// TIA Portal V17 export
// export: Created 2022-07-20T06:59:52.0228189Z, ExportSetting WithDefaults, DisplayName Totally Integrated Automation Portal, DisplayVersion V17, DisplayName TIA Portal Openness, DisplayVersion V17, DisplayName TIA Portal Version Control Interface, DisplayVersion V17, DisplayName SINAMICS Startdrive Advanced, DisplayVersion V17, DisplayName SINAMICS Startdrive G130, G150, S120, S150, SINAMICS MV, S210, DisplayVersion V17, DisplayName SINAMICS Startdrive G110M, G120, G120C, G120D, G120P, G115D, DisplayVersion V17, DisplayName STEP 7 Professional, DisplayVersion V17, DisplayName STEP 7 Safety, DisplayVersion V17, DisplayName WinCC Advanced, DisplayVersion V17
FUNCTION_BLOCK "FB10400_APCMotor"   // FB10400, LAD
{ S7_Optimized_Access := 'TRUE' }
VERSION : 0.1
// stored: AutoNumber false, IsIECCheckEnabled false, IsRetainMemResEnabled false, MemoryReserve 100, SetENOAutomatically false, UDAEnableTagReadback false
   VAR_INPUT
      ToAxis : TO_PositioningAxis;
      HomingSensor : Bool;
      RequestDirectHoming : Bool;
      RequestSensorHoming : Bool;
      RequestTorqueHoming : Bool;
      RequestGoToAbsolutePosition_1 : Bool;
      RequestGoToAbsolutePosition_2 : Bool;
      RequestGoToAbsolutePosition_3 : Bool;
      RequestGoToAbsolutePosition_4 : Bool;
      RequestGoToAbsolutePosition_5 : Bool;
      RequestGoToAbsolutePosition_6 : Bool;
      RequestGoToAbsolutePosition_7 : Bool;
      RequestGoToAbsolutePosition_8 : Bool;
      RequestGoToAbsolutePosition_9 : Bool;
      RequestGoToAbsolutePosition_10 : Bool;
      RequestGoToRelativePosition : Bool;
      RequestJogForward : Bool;
      RequestJogBackward : Bool;
      RequestStop : Bool;
      RequestFastStop : Bool;
      RequestAcknowledge : Bool;
      AbsolutePosition_1 : LReal;
      AbsolutePosition_2 : LReal;
      AbsolutePosition_3 : LReal;
      AbsolutePosition_4 : LReal;
      AbsolutePosition_5 : LReal;
      AbsolutePosition_6 : LReal;
      AbsolutePosition_7 : LReal;
      AbsolutePosition_8 : LReal;
      AbsolutePosition_9 : LReal;
      AbsolutePosition_10 : LReal;
      RelativePosition : Real;
   END_VAR
   VAR_OUTPUT
      AxisPositionningTooLong : Bool;
      HomingDone : Bool;
      ActualPosition_mm : LReal;
      IsInAbsolutePosition_1 { ExternalAccessible := 'False'; ExternalVisible := 'False'; ExternalWritable := 'False'} : Bool;
      IsInAbsolutePosition_2 { ExternalAccessible := 'False'; ExternalVisible := 'False'; ExternalWritable := 'False'} : Bool;
      IsInAbsolutePosition_3 { ExternalAccessible := 'False'; ExternalVisible := 'False'; ExternalWritable := 'False'} : Bool;
      IsInAbsolutePosition_4 { ExternalAccessible := 'False'; ExternalVisible := 'False'; ExternalWritable := 'False'} : Bool;
      IsInAbsolutePosition_5 { ExternalAccessible := 'False'; ExternalVisible := 'False'; ExternalWritable := 'False'} : Bool;
      IsInAbsolutePosition_6 { ExternalAccessible := 'False'; ExternalVisible := 'False'; ExternalWritable := 'False'} : Bool;
      IsInAbsolutePosition_7 { ExternalAccessible := 'False'; ExternalVisible := 'False'; ExternalWritable := 'False'} : Bool;
      IsInAbsolutePosition_8 { ExternalAccessible := 'False'; ExternalVisible := 'False'; ExternalWritable := 'False'} : Bool;
      IsInAbsolutePosition_9 { ExternalAccessible := 'False'; ExternalVisible := 'False'; ExternalWritable := 'False'} : Bool;
      IsInAbsolutePosition_10 { ExternalAccessible := 'False'; ExternalVisible := 'False'; ExternalWritable := 'False'} : Bool;
   END_VAR
   VAR_IN_OUT
      AxisStructure : "LAxisCtrl_Pos";
   END_VAR
   VAR
      i : USInt;
      MotorMovementStateDiagram : Int;
      Tolerence : Array[1..10] of Real;
      R_TRIG_DirectHoming : R_TRIG;
      R_TRIG_TorqueHoming { S7_SetPoint := 'True'} : R_TRIG;
      R_TRIG_SensorHoming { S7_SetPoint := 'True'} : R_TRIG;
      R_TRIG_SensorHomingDone { S7_SetPoint := 'True'} : R_TRIG;
      R_TRIG_RequestGoToAbsolutePosition { S7_SetPoint := 'True'} : Array[1..10] of R_TRIG;
      R_TRIG_RequestGoToRelativePosition { S7_SetPoint := 'True'} : R_TRIG;
      R_TRIG_JogForward { S7_SetPoint := 'True'} : R_TRIG;
      R_TRIG_JogBackward { S7_SetPoint := 'True'} : R_TRIG;
      F_TRIG_JogForward { S7_SetPoint := 'True'} : F_TRIG;
      F_TRIG_JogBackward { S7_SetPoint := 'True'} : F_TRIG;
      F_TRIG_AxisInError { S7_SetPoint := 'True'} : F_TRIG;
      TON_AxisCommandDone { S7_SetPoint := 'True'} : TON_TIME;
      TON_PositionningTooLong { S7_SetPoint := 'True'} : TON_TIME;
      MC_RESET_Instance { S7_SetPoint := 'True'} : MC_RESET;
      LAxisCtrl_PosAxis_Instance { S7_SetPoint := 'True'} : "LAxisCtrl_PosAxis";
      FB10401_MC_FixedStopHoming_APCFR_Instance { S7_SetPoint := 'True'} : "FB10401_MC_FixedStopHoming_APCFR";
      FB10403_MC_HomingOnSensor_Instance { S7_SetPoint := 'True'} : "FB10403_MC_HomingOnSensor";
      LAxisCtrl_GetAxisErrorWord_Instance { S7_SetPoint := 'True'} : "LAxisCtrl_GetAxisErrorWord";
      LAxisCtrl_GetAxisStatusWord_Instance { S7_SetPoint := 'True'} : "LAxisCtrl_GetAxisStatusWord";
   END_VAR
   VAR CONSTANT
      WAIT_FOR_MOTOR_REQUEST : Int := 0;
      DIRECT_HOMING : Int := 10;
      TORQUE_HOMING : Int := 20;
      SENSOR_HOMING : Int := 30;
      GO_TO_ABSOLUTE_POSITION_1 : Int := 40;
      GO_TO_ABSOLUTE_POSITION_2 : Int := 50;
      GO_TO_ABSOLUTE_POSITION_3 : Int := 60;
      GO_TO_ABSOLUTE_POSITION_4 : Int := 70;
      GO_TO_ABSOLUTE_POSITION_5 : Int := 80;
      GO_TO_ABSOLUTE_POSITION_6 : Int := 90;
      GO_TO_ABSOLUTE_POSITION_7 : Int := 100;
      GO_TO_ABSOLUTE_POSITION_8 : Int := 110;
      GO_TO_ABSOLUTE_POSITION_9 : Int := 120;
      GO_TO_ABSOLUTE_POSITION_10 : Int := 130;
      REQUEST_DONE : Int := 140;
   END_VAR
BEGIN

REGION Network 1 (SCL): First Scan
   IF "FirstScan" THEN
       #IsInAbsolutePosition_1 := FALSE;
       #IsInAbsolutePosition_2 := FALSE;
       #IsInAbsolutePosition_3 := FALSE;
       #IsInAbsolutePosition_4 := FALSE;
       #IsInAbsolutePosition_5 := FALSE;
       #IsInAbsolutePosition_6 := FALSE;
       #IsInAbsolutePosition_7 := FALSE;
       #IsInAbsolutePosition_8 := FALSE;
       #IsInAbsolutePosition_9 := FALSE;
       #IsInAbsolutePosition_10 := FALSE;
       #MotorMovementStateDiagram := #WAIT_FOR_MOTOR_REQUEST;
   END_IF;
END_REGION

REGION Network 2 (SCL): Edge Signals & Timer
   REGION EDGE SIGNALS
       #R_TRIG_DirectHoming(CLK := #RequestDirectHoming);
       #R_TRIG_TorqueHoming(CLK := #RequestTorqueHoming);
       #R_TRIG_SensorHoming(CLK := #RequestSensorHoming);
       #R_TRIG_SensorHomingDone(CLK := #AxisStructure.Out.SensorHomingDone);
       #R_TRIG_RequestGoToRelativePosition(CLK := #RequestGoToRelativePosition);
       #R_TRIG_RequestGoToAbsolutePosition[1](CLK := #RequestGoToAbsolutePosition_1);
       #R_TRIG_RequestGoToAbsolutePosition[2](CLK := #RequestGoToAbsolutePosition_2);
       #R_TRIG_RequestGoToAbsolutePosition[3](CLK := #RequestGoToAbsolutePosition_3);
       #R_TRIG_RequestGoToAbsolutePosition[4](CLK := #RequestGoToAbsolutePosition_4);
       #R_TRIG_RequestGoToAbsolutePosition[5](CLK := #RequestGoToAbsolutePosition_5);
       #R_TRIG_RequestGoToAbsolutePosition[6](CLK := #RequestGoToAbsolutePosition_6);
       #R_TRIG_RequestGoToAbsolutePosition[7](CLK := #RequestGoToAbsolutePosition_7);
       #R_TRIG_RequestGoToAbsolutePosition[8](CLK := #RequestGoToAbsolutePosition_8);
       #R_TRIG_RequestGoToAbsolutePosition[9](CLK := #RequestGoToAbsolutePosition_9);
       #R_TRIG_RequestGoToAbsolutePosition[10](CLK := #RequestGoToAbsolutePosition_10);
       #R_TRIG_JogForward(CLK := #RequestJogForward);
       #R_TRIG_JogBackward(CLK := #RequestJogBackward);

       #F_TRIG_AxisInError(CLK := #AxisStructure.Out.Error);
       #F_TRIG_JogForward(CLK := #RequestJogForward);
       #F_TRIG_JogBackward(CLK := #RequestJogBackward);
   END_REGION

   REGION TIMER
       #TON_AxisCommandDone(IN := #AxisStructure.Out.CommandDone,
                            PT := T#300ms);
       #TON_PositionningTooLong(IN := (#MotorMovementStateDiagram = #GO_TO_ABSOLUTE_POSITION_1) OR
                                (#MotorMovementStateDiagram = #GO_TO_ABSOLUTE_POSITION_2) OR
                                (#MotorMovementStateDiagram = #GO_TO_ABSOLUTE_POSITION_3) OR
                                (#MotorMovementStateDiagram = #GO_TO_ABSOLUTE_POSITION_4) OR
                                (#MotorMovementStateDiagram = #GO_TO_ABSOLUTE_POSITION_5) OR
                                (#MotorMovementStateDiagram = #GO_TO_ABSOLUTE_POSITION_6) OR
                                (#MotorMovementStateDiagram = #GO_TO_ABSOLUTE_POSITION_7) OR
                                (#MotorMovementStateDiagram = #GO_TO_ABSOLUTE_POSITION_8) OR
                                (#MotorMovementStateDiagram = #GO_TO_ABSOLUTE_POSITION_9) OR
                                (#MotorMovementStateDiagram = #GO_TO_ABSOLUTE_POSITION_10),
                                PT := T#30s);
   END_REGION
END_REGION

REGION Network 3 (SCL): Motor Parameters Management
   #AxisStructure.In.Config.posAbsolute.velocity := 25.0;
   #AxisStructure.In.Config.posAbsolute.acceleration := 100.0;
   #AxisStructure.In.Config.posAbsolute.deceleration := 100.0;
END_REGION

REGION Network 4: MC_Reset
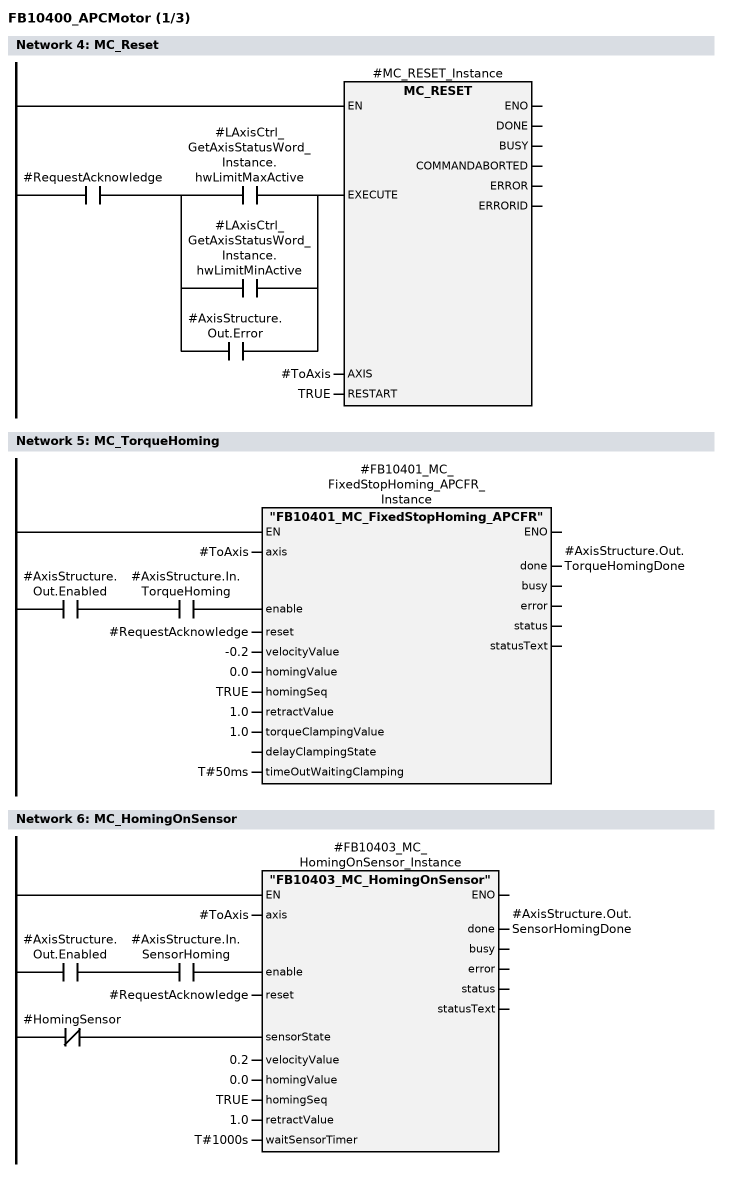
   RUNG wire#powerrail
      #MC_RESET_Instance.MC_RESET(Execute := wire#w2, Axis := #ToAxis, Restart := TRUE, Done =>, Busy =>, CommandAborted =>, Error =>, ErrorId =>)
   END_RUNG
   RUNG wire#powerrail
      Contact( #RequestAcknowledge )
      wire#w1
      Contact( #LAxisCtrl_GetAxisStatusWord_Instance.hwLimitMaxActive )
   END_RUNG wire#w2
   RUNG wire#w1
      Contact( #LAxisCtrl_GetAxisStatusWord_Instance.hwLimitMinActive )
   END_RUNG wire#w2
   RUNG wire#w1
      Contact( #AxisStructure.Out.Error )
   END_RUNG wire#w2
   // the same network as SCL:
   #MC_RESET_Instance(Execute := #RequestAcknowledge AND (#LAxisCtrl_GetAxisStatusWord_Instance.hwLimitMaxActive OR #LAxisCtrl_GetAxisStatusWord_Instance.hwLimitMinActive OR #AxisStructure.Out.Error),   // MC_RESET
                      Axis := #ToAxis,
                      Restart := TRUE);
END_REGION

REGION Network 5: MC_TorqueHoming
   RUNG wire#powerrail
      #FB10401_MC_FixedStopHoming_APCFR_Instance(enable := wire#w1, axis := #ToAxis, reset := #RequestAcknowledge, velocityValue := -0.2, homingValue := 0.0, homingSeq := TRUE, retractValue := 1.0, torqueClampingValue := 1.0, delayClampingState :=, timeOutWaitingClamping := T#50ms, done => #AxisStructure.Out.TorqueHomingDone, busy =>, error =>, status =>, statusText =>)
   END_RUNG
   RUNG wire#powerrail
      Contact( #AxisStructure.Out.Enabled )
      Contact( #AxisStructure.In.TorqueHoming )
   END_RUNG wire#w1
   // the same network as SCL:
   #FB10401_MC_FixedStopHoming_APCFR_Instance(axis := #ToAxis,   // "FB10401_MC_FixedStopHoming_APCFR"
                           enable := #AxisStructure.Out.Enabled AND #AxisStructure.In.TorqueHoming,
                           reset := #RequestAcknowledge,
                           velocityValue := -0.2,
                           homingValue := 0.0,
                           homingSeq := TRUE,
                           retractValue := 1.0,
                           torqueClampingValue := 1.0,
                           timeOutWaitingClamping := T#50ms,
                           done => #AxisStructure.Out.TorqueHomingDone);
END_REGION

REGION Network 6: MC_HomingOnSensor
   RUNG wire#powerrail
      #FB10403_MC_HomingOnSensor_Instance(enable := wire#w1, sensorState := wire#w2, axis := #ToAxis, reset := #RequestAcknowledge, velocityValue := 0.2, homingValue := 0.0, homingSeq := TRUE, retractValue := 1.0, waitSensorTimer := T#1000s, done => #AxisStructure.Out.SensorHomingDone, busy =>, error =>, status =>, statusText =>)
   END_RUNG
   RUNG wire#powerrail
      Contact( #AxisStructure.Out.Enabled )
      Contact( #AxisStructure.In.SensorHoming )
   END_RUNG wire#w1
   RUNG wire#powerrail
      I_Contact( #HomingSensor )
   END_RUNG wire#w2
   // the same network as SCL:
   #FB10403_MC_HomingOnSensor_Instance(axis := #ToAxis,   // "FB10403_MC_HomingOnSensor"
                           enable := #AxisStructure.Out.Enabled AND #AxisStructure.In.SensorHoming,
                           reset := #RequestAcknowledge,
                           sensorState := NOT #HomingSensor,
                           velocityValue := 0.2,
                           homingValue := 0.0,
                           homingSeq := TRUE,
                           retractValue := 1.0,
                           waitSensorTimer := T#1000s,
                           done => #AxisStructure.Out.SensorHomingDone);
END_REGION

REGION Network 7: Axis Manager
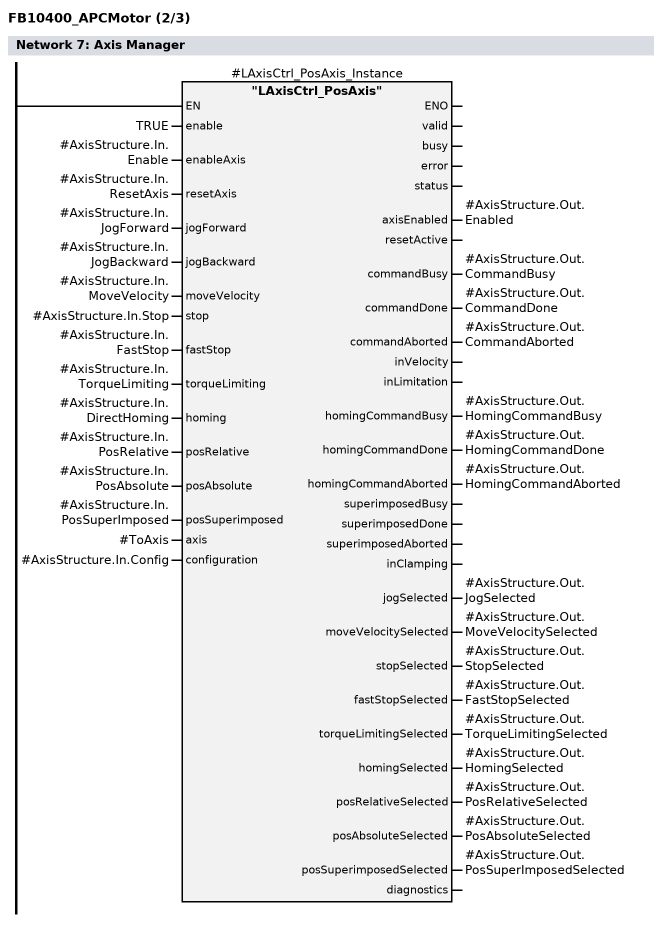
   RUNG wire#powerrail
      #LAxisCtrl_PosAxis_Instance(enable := TRUE, enableAxis := #AxisStructure.In.Enable, resetAxis := #AxisStructure.In.ResetAxis, jogForward := #AxisStructure.In.JogForward, jogBackward := #AxisStructure.In.JogBackward, moveVelocity := #AxisStructure.In.MoveVelocity, stop := #AxisStructure.In.Stop, fastStop := #AxisStructure.In.FastStop, torqueLimiting := #AxisStructure.In.TorqueLimiting, homing := #AxisStructure.In.DirectHoming, posRelative := #AxisStructure.In.PosRelative, posAbsolute := #AxisStructure.In.PosAbsolute, posSuperimposed := #AxisStructure.In.PosSuperImposed, axis := #ToAxis, configuration := #AxisStructure.In.Config, valid =>, busy =>, error =>, status =>, axisEnabled => #AxisStructure.Out.Enabled, resetActive =>, commandBusy => #AxisStructure.Out.CommandBusy, commandDone => #AxisStructure.Out.CommandDone, commandAborted => #AxisStructure.Out.CommandAborted, inVelocity =>, inLimitation =>, homingCommandBusy => #AxisStructure.Out.HomingCommandBusy, homingCommandDone => #AxisStructure.Out.HomingCommandDone, homingCommandAborted => #AxisStructure.Out.HomingCommandAborted, superimposedBusy =>, superimposedDone =>, superimposedAborted =>, inClamping =>, jogSelected => #AxisStructure.Out.JogSelected, moveVelocitySelected => #AxisStructure.Out.MoveVelocitySelected, stopSelected => #AxisStructure.Out.StopSelected, fastStopSelected => #AxisStructure.Out.FastStopSelected, torqueLimitingSelected => #AxisStructure.Out.TorqueLimitingSelected, homingSelected => #AxisStructure.Out.HomingSelected, posRelativeSelected => #AxisStructure.Out.PosRelativeSelected, posAbsoluteSelected => #AxisStructure.Out.PosAbsoluteSelected, posSuperimposedSelected => #AxisStructure.Out.PosSuperImposedSelected, diagnostics =>)
   END_RUNG
   // the same network as SCL:
   #LAxisCtrl_PosAxis_Instance(enable := TRUE,   // "LAxisCtrl_PosAxis"
                           enableAxis := #AxisStructure.In.Enable,
                           resetAxis := #AxisStructure.In.ResetAxis,
                           jogForward := #AxisStructure.In.JogForward,
                           jogBackward := #AxisStructure.In.JogBackward,
                           moveVelocity := #AxisStructure.In.MoveVelocity,
                           stop := #AxisStructure.In.Stop,
                           fastStop := #AxisStructure.In.FastStop,
                           torqueLimiting := #AxisStructure.In.TorqueLimiting,
                           homing := #AxisStructure.In.DirectHoming,
                           posRelative := #AxisStructure.In.PosRelative,
                           posAbsolute := #AxisStructure.In.PosAbsolute,
                           posSuperimposed := #AxisStructure.In.PosSuperImposed,
                           axis := #ToAxis,
                           configuration := #AxisStructure.In.Config,
                           axisEnabled => #AxisStructure.Out.Enabled,
                           commandBusy => #AxisStructure.Out.CommandBusy,
                           commandDone => #AxisStructure.Out.CommandDone,
                           commandAborted => #AxisStructure.Out.CommandAborted,
                           homingCommandBusy => #AxisStructure.Out.HomingCommandBusy,
                           homingCommandDone => #AxisStructure.Out.HomingCommandDone,
                           homingCommandAborted => #AxisStructure.Out.HomingCommandAborted,
                           jogSelected => #AxisStructure.Out.JogSelected,
                           moveVelocitySelected => #AxisStructure.Out.MoveVelocitySelected,
                           stopSelected => #AxisStructure.Out.StopSelected,
                           fastStopSelected => #AxisStructure.Out.FastStopSelected,
                           torqueLimitingSelected => #AxisStructure.Out.TorqueLimitingSelected,
                           homingSelected => #AxisStructure.Out.HomingSelected,
                           posRelativeSelected => #AxisStructure.Out.PosRelativeSelected,
                           posAbsoluteSelected => #AxisStructure.Out.PosAbsoluteSelected,
                           posSuperimposedSelected => #AxisStructure.Out.PosSuperImposedSelected);
END_REGION

REGION Network 8: Motor Error Word and Status Word
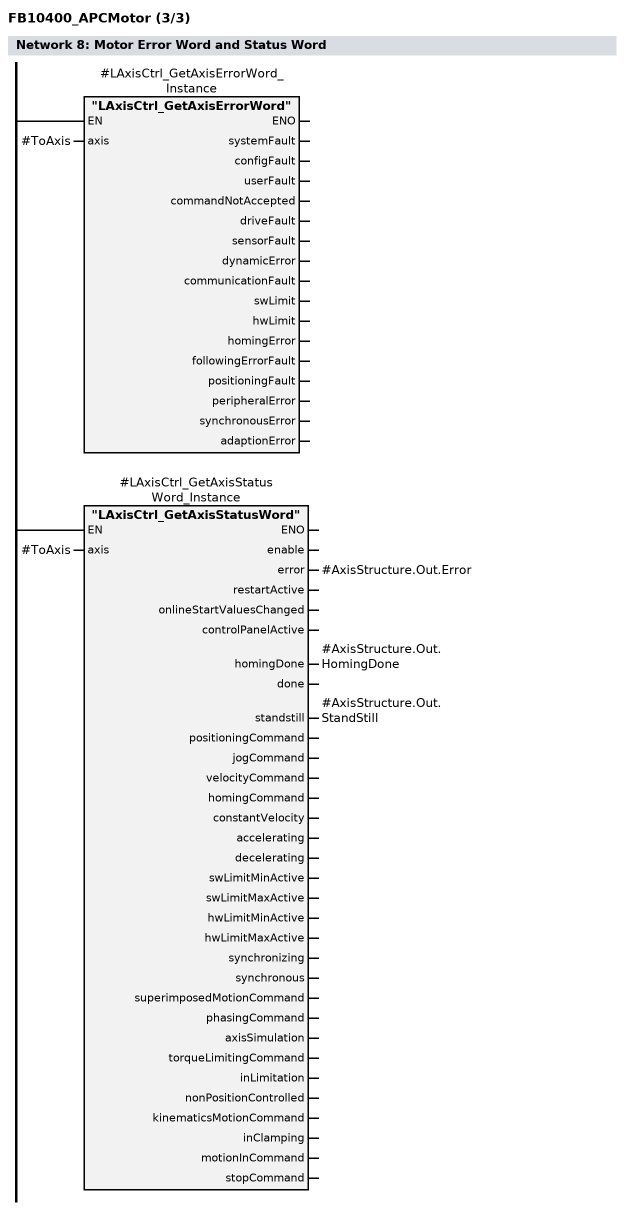
   RUNG wire#powerrail
      #LAxisCtrl_GetAxisErrorWord_Instance(axis := #ToAxis, systemFault =>, configFault =>, userFault =>, commandNotAccepted =>, driveFault =>, sensorFault =>, dynamicError =>, communicationFault =>, swLimit =>, hwLimit =>, homingError =>, followingErrorFault =>, positioningFault =>, peripheralError =>, synchronousError =>, adaptionError =>)
   END_RUNG
   RUNG wire#powerrail
      #LAxisCtrl_GetAxisStatusWord_Instance(axis := #ToAxis, enable =>, error => #AxisStructure.Out.Error, restartActive =>, onlineStartValuesChanged =>, controlPanelActive =>, homingDone => #AxisStructure.Out.HomingDone, done =>, standstill => #AxisStructure.Out.StandStill, positioningCommand =>, jogCommand =>, velocityCommand =>, homingCommand =>, constantVelocity =>, accelerating =>, decelerating =>, swLimitMinActive =>, swLimitMaxActive =>, hwLimitMinActive =>, hwLimitMaxActive =>, synchronizing =>, synchronous =>, superimposedMotionCommand =>, phasingCommand =>, axisSimulation =>, torqueLimitingCommand =>, inLimitation =>, nonPositionControlled =>, kinematicsMotionCommand =>, inClamping =>, motionInCommand =>, stopCommand =>)
   END_RUNG
   // the same network as SCL:
   #LAxisCtrl_GetAxisErrorWord_Instance(axis := #ToAxis);   // "LAxisCtrl_GetAxisErrorWord"
   #LAxisCtrl_GetAxisStatusWord_Instance(axis := #ToAxis,   // "LAxisCtrl_GetAxisStatusWord"
                           error => #AxisStructure.Out.Error,
                           homingDone => #AxisStructure.Out.HomingDone,
                           standstill => #AxisStructure.Out.StandStill);
END_REGION

REGION Network 9 (SCL): Motor Movement Management
   IF #RequestStop THEN
       #AxisStructure.In.TorqueHoming := FALSE;
       #AxisStructure.In.DirectHoming := FALSE;
       #AxisStructure.In.SensorHoming := FALSE;
       #AxisStructure.In.PosAbsolute := FALSE;
       #AxisStructure.In.Enable := FALSE;
       #MotorMovementStateDiagram := #WAIT_FOR_MOTOR_REQUEST;
   END_IF;

   CASE #MotorMovementStateDiagram OF
       #WAIT_FOR_MOTOR_REQUEST:
           IF #R_TRIG_DirectHoming.Q THEN
               #AxisStructure.In.TorqueHoming := FALSE;
               #AxisStructure.In.DirectHoming := FALSE;
               #AxisStructure.In.SensorHoming := FALSE;
               #AxisStructure.In.PosAbsolute := FALSE;
               #MotorMovementStateDiagram := #DIRECT_HOMING;
           ELSIF #R_TRIG_TorqueHoming.Q THEN
               #AxisStructure.In.TorqueHoming := FALSE;
               #AxisStructure.In.DirectHoming := FALSE;
               #AxisStructure.In.SensorHoming := FALSE;
               #AxisStructure.In.PosAbsolute := FALSE;
               #MotorMovementStateDiagram := #TORQUE_HOMING;
           ELSIF #R_TRIG_SensorHoming.Q THEN
               #HomingDone := FALSE;
               #AxisStructure.In.TorqueHoming := FALSE;
               #AxisStructure.In.DirectHoming := FALSE;
               #AxisStructure.In.SensorHoming := FALSE;
               #AxisStructure.In.PosAbsolute := FALSE;
               #MotorMovementStateDiagram := #SENSOR_HOMING;
           ELSIF #R_TRIG_RequestGoToAbsolutePosition[1].Q THEN
               #AxisStructure.In.PosAbsolute := FALSE;
               #MotorMovementStateDiagram := #GO_TO_ABSOLUTE_POSITION_1;
           ELSIF #R_TRIG_RequestGoToAbsolutePosition[2].Q THEN
               #AxisStructure.In.PosAbsolute := FALSE;
               #MotorMovementStateDiagram := #GO_TO_ABSOLUTE_POSITION_2;
           ELSIF #R_TRIG_RequestGoToAbsolutePosition[3].Q THEN
               #AxisStructure.In.PosAbsolute := FALSE;
               #MotorMovementStateDiagram := #GO_TO_ABSOLUTE_POSITION_3;
           ELSIF #R_TRIG_RequestGoToAbsolutePosition[4].Q THEN
               #AxisStructure.In.PosAbsolute := FALSE;
               #MotorMovementStateDiagram := #GO_TO_ABSOLUTE_POSITION_4;
           ELSIF #R_TRIG_RequestGoToAbsolutePosition[5].Q THEN
               #AxisStructure.In.PosAbsolute := FALSE;
               #MotorMovementStateDiagram := #GO_TO_ABSOLUTE_POSITION_5;
           ELSIF #R_TRIG_RequestGoToAbsolutePosition[6].Q THEN
               #AxisStructure.In.PosAbsolute := FALSE;
               #MotorMovementStateDiagram := #GO_TO_ABSOLUTE_POSITION_6;
           ELSIF #R_TRIG_RequestGoToAbsolutePosition[7].Q THEN
               #AxisStructure.In.PosAbsolute := FALSE;
               #MotorMovementStateDiagram := #GO_TO_ABSOLUTE_POSITION_7;
           ELSIF #R_TRIG_RequestGoToAbsolutePosition[8].Q THEN
               #AxisStructure.In.PosAbsolute := FALSE;
               #MotorMovementStateDiagram := #GO_TO_ABSOLUTE_POSITION_8;
           ELSIF #R_TRIG_RequestGoToAbsolutePosition[9].Q THEN
               #AxisStructure.In.PosAbsolute := FALSE;
               #MotorMovementStateDiagram := #GO_TO_ABSOLUTE_POSITION_9;
           ELSIF #R_TRIG_RequestGoToAbsolutePosition[10].Q THEN
               #AxisStructure.In.PosAbsolute := FALSE;
               #MotorMovementStateDiagram := #GO_TO_ABSOLUTE_POSITION_10;
           ELSE
               #AxisStructure.In.TorqueHoming := FALSE;
               #AxisStructure.In.DirectHoming := FALSE;
               #AxisStructure.In.SensorHoming := FALSE;
               #AxisStructure.In.PosAbsolute := FALSE;
           END_IF;
       #DIRECT_HOMING:
           #AxisStructure.In.Config.homing.position := 0.0;
           #AxisStructure.In.Config.homing.extendedMode := -1;
           #AxisStructure.In.Config.homing.mode := 7;
           #AxisStructure.In.DirectHoming := TRUE;
           IF #AxisStructure.Out.HomingCommandDone THEN
               #AxisStructure.In.DirectHoming := FALSE;
               #MotorMovementStateDiagram := #REQUEST_DONE;
           END_IF;
       #TORQUE_HOMING:
           IF #AxisStructure.Out.Enabled THEN
               #AxisStructure.In.TorqueHoming := TRUE;
               IF #AxisStructure.Out.TorqueHomingDone THEN
                   #AxisStructure.In.Enable := FALSE;
                   #AxisStructure.In.TorqueHoming := FALSE;

                   #MotorMovementStateDiagram := #REQUEST_DONE;
               END_IF;
           ELSE
               #AxisStructure.In.Enable := TRUE;
           END_IF;
       #SENSOR_HOMING:
           IF #AxisStructure.Out.Enabled THEN
               #AxisStructure.In.SensorHoming := TRUE;
               IF #R_TRIG_SensorHomingDone.Q THEN
                   #AxisStructure.In.Enable := FALSE;
                   #AxisStructure.In.SensorHoming := FALSE;
                   #MotorMovementStateDiagram := #REQUEST_DONE;
               END_IF;
           ELSE
               #AxisStructure.In.Enable := TRUE;
           END_IF;
       #GO_TO_ABSOLUTE_POSITION_1:
           IF #AxisStructure.Out.Enabled AND #AxisStructure.Out.HomingDone THEN
               #AxisStructure.In.Config.posAbsolute.position := #AbsolutePosition_1;
               #AxisStructure.In.PosAbsolute := TRUE;
               IF #TON_AxisCommandDone.Q THEN
                   #AxisStructure.In.PosAbsolute := FALSE;
                   #AxisStructure.In.Enable := FALSE;
                   #MotorMovementStateDiagram := #REQUEST_DONE;
               END_IF;
           ELSE
               #AxisStructure.In.Enable := TRUE;
           END_IF;
       #GO_TO_ABSOLUTE_POSITION_2:
           IF #AxisStructure.Out.Enabled AND #AxisStructure.Out.HomingDone THEN
               #AxisStructure.In.Config.posAbsolute.position := #AbsolutePosition_2;
               #AxisStructure.In.PosAbsolute := TRUE;
               IF #TON_AxisCommandDone.Q THEN
                   #AxisStructure.In.PosAbsolute := FALSE;
                   #AxisStructure.In.Enable := FALSE;
                   #MotorMovementStateDiagram := #REQUEST_DONE;
               END_IF;
           ELSE
               #AxisStructure.In.Enable := TRUE;
           END_IF;
       #GO_TO_ABSOLUTE_POSITION_3:
           IF #AxisStructure.Out.Enabled AND #AxisStructure.Out.HomingDone THEN
               #AxisStructure.In.Config.posAbsolute.position := #AbsolutePosition_3;
               #AxisStructure.In.PosAbsolute := TRUE;
               IF #TON_AxisCommandDone.Q THEN
                   #AxisStructure.In.PosAbsolute := FALSE;
                   #AxisStructure.In.Enable := FALSE;
                   #MotorMovementStateDiagram := #REQUEST_DONE;
               END_IF;
           ELSE
               #AxisStructure.In.Enable := TRUE;
           END_IF;
       #GO_TO_ABSOLUTE_POSITION_4:
           IF #AxisStructure.Out.Enabled AND #AxisStructure.Out.HomingDone THEN
               #AxisStructure.In.Config.posAbsolute.position := #AbsolutePosition_4;
               #AxisStructure.In.PosAbsolute := TRUE;
               IF #TON_AxisCommandDone.Q THEN
                   #AxisStructure.In.PosAbsolute := FALSE;
                   #AxisStructure.In.Enable := FALSE;
                   #MotorMovementStateDiagram := #REQUEST_DONE;
               END_IF;
           ELSE
               #AxisStructure.In.Enable := TRUE;
           END_IF;
       #GO_TO_ABSOLUTE_POSITION_5:
           IF #AxisStructure.Out.Enabled AND #AxisStructure.Out.HomingDone THEN
               #AxisStructure.In.Config.posAbsolute.position := #AbsolutePosition_5;
               #AxisStructure.In.PosAbsolute := TRUE;
               IF #TON_AxisCommandDone.Q THEN
                   #AxisStructure.In.PosAbsolute := FALSE;
                   #AxisStructure.In.Enable := FALSE;
                   #MotorMovementStateDiagram := #REQUEST_DONE;
               END_IF;
           ELSE
               #AxisStructure.In.Enable := TRUE;
           END_IF;
       #GO_TO_ABSOLUTE_POSITION_6:
           IF #AxisStructure.Out.Enabled AND #AxisStructure.Out.HomingDone THEN
               #AxisStructure.In.Config.posAbsolute.position := #AbsolutePosition_6;
               #AxisStructure.In.PosAbsolute := TRUE;
               IF #TON_AxisCommandDone.Q THEN
                   #IsInAbsolutePosition_6 := TRUE;
                   #AxisStructure.In.PosAbsolute := FALSE;
                   #AxisStructure.In.Enable := FALSE;
                   #MotorMovementStateDiagram := #REQUEST_DONE;
               END_IF;
           ELSE
               #AxisStructure.In.Enable := TRUE;
           END_IF;
       #GO_TO_ABSOLUTE_POSITION_7:
           IF #AxisStructure.Out.Enabled AND #AxisStructure.Out.HomingDone THEN
               #AxisStructure.In.Config.posAbsolute.position := #AbsolutePosition_7;
               #AxisStructure.In.PosAbsolute := TRUE;
               IF #TON_AxisCommandDone.Q THEN
                   #AxisStructure.In.PosAbsolute := FALSE;
                   #AxisStructure.In.Enable := FALSE;
                   #MotorMovementStateDiagram := #REQUEST_DONE;
               END_IF;
           ELSE
               #AxisStructure.In.Enable := TRUE;
           END_IF;
       #GO_TO_ABSOLUTE_POSITION_8:
           IF #AxisStructure.Out.Enabled AND #AxisStructure.Out.HomingDone THEN
               #AxisStructure.In.Config.posAbsolute.position := #AbsolutePosition_8;
               #AxisStructure.In.PosAbsolute := TRUE;
               IF #TON_AxisCommandDone.Q THEN
                   #AxisStructure.In.PosAbsolute := FALSE;
                   #AxisStructure.In.Enable := FALSE;
                   #MotorMovementStateDiagram := #REQUEST_DONE;
               END_IF;
           ELSE
               #AxisStructure.In.Enable := TRUE;
           END_IF;
       #GO_TO_ABSOLUTE_POSITION_9:
           IF #AxisStructure.Out.Enabled AND #AxisStructure.Out.HomingDone THEN
               #AxisStructure.In.Config.posAbsolute.position := #AbsolutePosition_9;
               #AxisStructure.In.PosAbsolute := TRUE;
               IF #TON_AxisCommandDone.Q THEN
                   #AxisStructure.In.PosAbsolute := FALSE;
                   #AxisStructure.In.Enable := FALSE;
                   #MotorMovementStateDiagram := #REQUEST_DONE;
               END_IF;
           ELSE
               #AxisStructure.In.Enable := TRUE;
           END_IF;
       #GO_TO_ABSOLUTE_POSITION_10:
           IF #AxisStructure.Out.Enabled AND #AxisStructure.Out.HomingDone THEN
               #AxisStructure.In.Config.posAbsolute.position := #AbsolutePosition_10;
               #AxisStructure.In.PosAbsolute := TRUE;
               IF #TON_AxisCommandDone.Q THEN
                   #AxisStructure.In.PosAbsolute := FALSE;
                   #AxisStructure.In.Enable := FALSE;
                   #MotorMovementStateDiagram := #REQUEST_DONE;
               END_IF;
           ELSE
               #AxisStructure.In.Enable := TRUE;
           END_IF;
       #REQUEST_DONE:
           #MotorMovementStateDiagram := #WAIT_FOR_MOTOR_REQUEST;
   END_CASE;
END_REGION

REGION Network 10 (SCL): Motor States Management
   IF #AxisStructure.Out.HomingDone THEN
       REGION Tolerence Value Management
           IF #AbsolutePosition_1 = 0.0 THEN
               #Tolerence[1] := 0.1;
           ELSE
               #Tolerence[1] := 0.05;
           END_IF;

           IF #AbsolutePosition_2 = 0.0 THEN
               #Tolerence[2] := 0.1;
           ELSE
               #Tolerence[2] := 0.05;
           END_IF;

           IF #AbsolutePosition_3 = 0.0 THEN
               #Tolerence[3] := 0.1;
           ELSE
               #Tolerence[3] := 0.05;
           END_IF;

           IF #AbsolutePosition_4 = 0.0 THEN
               #Tolerence[4] := 0.1;
           ELSE
               #Tolerence[4] := 0.05;
           END_IF;

           IF #AbsolutePosition_5 = 0.0 THEN
               #Tolerence[5] := 0.1;
           ELSE
               #Tolerence[5] := 0.05;
           END_IF;

           IF #AbsolutePosition_6 = 0.0 THEN
               #Tolerence[6] := 0.1;
           ELSE
               #Tolerence[6] := 0.05;
           END_IF;

           IF #AbsolutePosition_7 = 0.0 THEN
               #Tolerence[7] := 0.1;
           ELSE
               #Tolerence[7] := 0.05;
           END_IF;

           IF #AbsolutePosition_8 = 0.0 THEN
               #Tolerence[8] := 0.1;
           ELSE
               #Tolerence[8] := 0.05;
           END_IF;

           IF #AbsolutePosition_9 = 0.0 THEN
               #Tolerence[9] := 0.1;
           ELSE
               #Tolerence[9] := 0.05;
           END_IF;

           IF #AbsolutePosition_10 = 0.0 THEN
               #Tolerence[10] := 0.1;
           ELSE
               #Tolerence[10] := 0.05;
           END_IF;
       END_REGION

       REGION Position Test Management
           #IsInAbsolutePosition_1 := "FC10021_TolerenceRelation"(X := #ToAxis.ActualPosition, Y := #AbsolutePosition_1, Tolerance := #Tolerence[1]);
           #IsInAbsolutePosition_2 := "FC10021_TolerenceRelation"(X := #ToAxis.ActualPosition, Y := #AbsolutePosition_2, Tolerance := #Tolerence[2]);
           #IsInAbsolutePosition_3 := "FC10021_TolerenceRelation"(X := #ToAxis.ActualPosition, Y := #AbsolutePosition_3, Tolerance := #Tolerence[3]);
           #IsInAbsolutePosition_4 := "FC10021_TolerenceRelation"(X := #ToAxis.ActualPosition, Y := #AbsolutePosition_4, Tolerance := #Tolerence[4]);
           #IsInAbsolutePosition_5 := "FC10021_TolerenceRelation"(X := #ToAxis.ActualPosition, Y := #AbsolutePosition_5, Tolerance := #Tolerence[5]);
           #IsInAbsolutePosition_6 := "FC10021_TolerenceRelation"(X := #ToAxis.ActualPosition, Y := #AbsolutePosition_6, Tolerance := #Tolerence[6]);
           #IsInAbsolutePosition_7 := "FC10021_TolerenceRelation"(X := #ToAxis.ActualPosition, Y := #AbsolutePosition_7, Tolerance := #Tolerence[7]);
           #IsInAbsolutePosition_8 := "FC10021_TolerenceRelation"(X := #ToAxis.ActualPosition, Y := #AbsolutePosition_8, Tolerance := #Tolerence[8]);
           #IsInAbsolutePosition_9 := "FC10021_TolerenceRelation"(X := #ToAxis.ActualPosition, Y := #AbsolutePosition_9, Tolerance := #Tolerence[9]);
           #IsInAbsolutePosition_10 := "FC10021_TolerenceRelation"(X := #ToAxis.ActualPosition, Y := #AbsolutePosition_10, Tolerance := #Tolerence[10]);
       END_REGION
   ELSE
       #IsInAbsolutePosition_1 := FALSE;
       #IsInAbsolutePosition_2 := FALSE;
       #IsInAbsolutePosition_3 := FALSE;
       #IsInAbsolutePosition_4 := FALSE;
       #IsInAbsolutePosition_5 := FALSE;
       #IsInAbsolutePosition_6 := FALSE;
       #IsInAbsolutePosition_7 := FALSE;
       #IsInAbsolutePosition_8 := FALSE;
       #IsInAbsolutePosition_9 := FALSE;
       #IsInAbsolutePosition_10 := FALSE;
   END_IF;
   #HomingDone := #AxisStructure.Out.SensorHomingDone;
   #ActualPosition_mm := #ToAxis.ActualPosition;
END_REGION

REGION Network 11 (SCL): Motor Error Management
   //Error Management
   IF #AxisStructure.Out.Error OR #TON_PositionningTooLong.Q THEN
       #MotorMovementStateDiagram := #WAIT_FOR_MOTOR_REQUEST;
       #AxisStructure.In.Enable := FALSE;
       #AxisStructure.In.ResetAxis := FALSE;
       IF #TON_PositionningTooLong.Q THEN
           #AxisPositionningTooLong := TRUE;
       END_IF;
   END_IF;

   //Acknowledge Management
   IF #AxisStructure.Out.Error AND #RequestAcknowledge THEN
       #AxisStructure.In.ResetAxis := TRUE;
   END_IF;
   IF #F_TRIG_AxisInError.Q THEN
       #AxisStructure.In.ResetAxis := FALSE;
   END_IF;
   IF #RequestAcknowledge THEN
       #AxisPositionningTooLong := FALSE;
   END_IF;
END_REGION
END_FUNCTION_BLOCK
